{attribute 'qualified_only'}
{attribute 'strict'}
TYPE Saw :
(
	on := 0,
	off 
);
END_TYPE

(* stored: Version 1.1.0.1, ProductVersion 3.1.4022.12
   DUT Saw: Id {57bee488-8426-4ae4-ab68-7cf672f8e858} *)
